// TwinCAT 3 PLC project Untitled1
// ProgramVersion: 3.1.4026.1+972e9c44872ad038b353624a861fd7e3244e9f75
// libraries:
//   Tc2_Standard, * (Beckhoff Automation GmbH)
//   Tc2_System, * (Beckhoff Automation GmbH)
//   Tc2_Utilities, * (Beckhoff Automation GmbH)
// project tree:
//   FolderControl/ E_FolderControlState.TcDUT, FB_FolderControl.TcPOU
//   FileWriter/ E_FileWriteState.TcDUT, FB_FileControl.TcPOU
//   / PlcTask.TcTTO
//   POUs/ MAIN.TcPOU
// real-time tasks:
//   TASK PlcTask: cycle T#10ms, priority 20, ADS port 350

CONFIGURATION Untitled1
    RESOURCE PLC ON TwinCAT3
        TASK PlcTask(INTERVAL := T#10ms, PRIORITY := 20);
        PROGRAM MAIN WITH PlcTask : MAIN;
    END_RESOURCE
END_CONFIGURATION

// ---- FolderControl/E_FolderControlState.TcDUT
{attribute 'qualified_only'}
{attribute 'strict'}
{attribute 'to_string'}
TYPE E_FolderControlState :
(
	init := 0,
	ReadyFindFolder := 10,
	FindFolder := 20,
	ReadyForCreateFolder := 100,
	CreateFolder := 110,
	Error := 999
);
END_TYPE

// ---- FileWriter/E_FileWriteState.TcDUT
{attribute 'qualified_only'}
{attribute 'strict'}
{attribute 'to_string'}
TYPE E_FileWriteState :
(
	init := 0,
	ReadyFileCreate := 5,
	FileOpen := 10, 
	FileWrite := 20, 
	FileClose := 30, 
	Error := 999
);
END_TYPE

// ---- POUs/MAIN.TcPOU
PROGRAM MAIN
VAR
	fbFolderControl : FB_FolderControl;
	sPath : T_MaxString := 'C:\Test\test2\test3';
	sFile : STRING;
	bStart: BOOL;
	bCheck: BOOL;
	
	step : INT;
	fbFileControl : FB_FileControl;
	sTest : T_MaxString;
END_VAR


IF bStart THEN
	bStart := FALSE;
	fbFolderControl.CreateFolder(sPath);
END_IF
IF bCheck THEN
	bCheck := FALSE;
	fbFolderControl.CheckFolder(sPath);
END_IF

fbFolderCOntrol.CyclicLogic();

CASE step OF
	0:
		;
	10:
		fbFileControl.OverwriteFile(sPath,ADR(sTest),LEN(sTest));
		step := 0;
	20:
		fbFileControl.AppendwriteFile(sPath,ADR(sTest),LEN(sTest));
		step := 0;
END_CASE
fbFileControl.CyclicLogit();

END_PROGRAM

// ---- FolderControl/FB_FolderControl.TcPOU
FUNCTION_BLOCK FB_FolderControl
VAR
	eState : E_FolderControlState;
	fbEnumFindFileEntry : FB_EnumFindFileEntry;
	fbCreateDir : FB_CreateDir;
	_CreateFolderPath : T_MAXSTRING;
	_CheckFolderPath : T_MAXSTRING;
	_FolderExist : BOOL;
	
	_Error : BOOL;
	_ErrorID : UDINT;
	_ErrorState : STRING(50);
	_AmsNetID : T_AmsNetID;
END_VAR

PROPERTY AmsNetId : T_AmsNetId
GET
AmsNetId := _AmsNetId;
END_GET
SET
_AmsNetId := AmsNetId;
END_SET
END_PROPERTY

{attribute 'monitoring':='call'}
PROPERTY Busy : BOOL
GET
Busy := NOT (eState = 0 OR eState = E_FolderControlState.Error);
END_GET
END_PROPERTY

METHOD CheckFolder : BOOL
VAR_INPUT
	sPath : T_MAXSTRING;
END_VAR
VAR
	i : INT;
END_VAR
IF Busy THEN
	RETURN;
END_IF
ResetStatus();

eState := E_FolderControlState.ReadyFindFolder;

MEMSET(ADR(_CheckFolderPath), 0, SIZEOF(_CheckFolderPath));

IF RIGHT(sPath,1) = '/' OR RIGHT(sPath,1) = '\' THEN
	sPath := Delete(sPath,1,LEN(sPath));
END_IF

FOR i:=0 TO LEN(sPath) BY 1 DO
	IF sPath[i] = 47 THEN 	// '/'
		_CheckFolderPath[i] := 92; 	// '\'
	ELSE
		_CheckFolderPath[i] := sPath[i];
	END_IF	
END_FOR

CheckFolder := TRUE;
END_METHOD

METHOD CreateFolder : BOOL
VAR_INPUT
	sPath : T_MAXSTRING;
END_VAR
VAR
	i : INT;
END_VAR
(*
	It only can create one more subfolder
	폴더 한번에 한개만 생성가능 즉, C:\Test\Test1\Test2 를 생성하고자 할때 Test1 폴더가 없으면 생성 불가
*)
IF Busy THEN
	RETURN;
END_IF
ResetStatus();

eState := E_FolderControlState.ReadyForCreateFolder;

MEMSET(ADR(_CreateFolderPath), 0, SIZEOF(_CreateFolderPath));

IF RIGHT(sPath,1) = '/' OR RIGHT(sPath,1) = '\' THEN
	sPath := Delete(sPath,1,LEN(sPath));
END_IF

FOR i:=0 TO LEN(sPath) BY 1 DO
	IF sPath[i] = 47 THEN 	// '/'
		_CreateFolderPath[i] := 92; 	// '\'
	ELSE
		_CreateFolderPath[i] := sPath[i];
	END_IF	
END_FOR

CreateFolder := TRUE;
END_METHOD

METHOD CyclicLogic
VAR_INPUT
END_VAR
CASE eState OF
	E_FolderControlState.init:
		;
		
	E_FolderControlState.ReadyFindFolder:
		fbEnumFindFileEntry(bExecute:= FALSE);
		fbEnumFindFileEntry.eCmd := E_EnumCmdType.eEnumCmd_First;
		_FolderExist := FALSE;
		eState := E_FolderControlState.FindFolder;
	
	E_FolderControlState.FindFolder:
		fbEnumFindFileEntry( 
			sPathName:= _CheckFolderPath, 
			bExecute:= TRUE);
		IF NOT fbEnumFindFileEntry.bBusy THEN
			IF fbEnumFindFileEntry.stFindFile.fileAttributes.bDirectory THEN
				_FolderExist := TRUE;
				eState := E_FolderControlState.init;
			END_IF
		END_IF
		
	E_FolderControlState.ReadyForCreateFolder:
		fbCreateDir(bExecute:= FALSE);
		eState := E_FolderControlState.CreateFolder;
		
	E_FolderControlState.CreateFolder:
		fbCreateDir(
			sNetId:= , 
			sPathName:= _CreateFolderPath,
			ePath:= E_OpenPath.PATH_GENERIC, 
			bExecute:= TRUE, 
			tTimeout:= , 
			bBusy=> , 
			bError=> , 
			nErrId=> );
		IF NOT fbCreateDir.bBusy THEN
			IF fbCreateDir.bError THEN
				_ErrorState := TO_STRING(E_FolderControlState.CreateFolder);
				eState := E_FolderControlState.Error;
				_ErrorID := fbCreateDir.nErrId;
			ELSE
				eState := E_FolderControlState.init;
			END_IF
		END_IF
	
	E_FolderControlState.Error:
		_Error := TRUE;
END_CASE
END_METHOD

{attribute 'monitoring':='variable'}
PROPERTY Error : BOOL
GET
Error := _Error;
END_GET
END_PROPERTY

{attribute 'monitoring':='variable'}
PROPERTY ErrorID : UDINT
GET
ErrorID := _ErrorID;
END_GET
END_PROPERTY

PROPERTY isFolderExist : BOOL
GET
isFolderExist := _FolderExist;
END_GET
END_PROPERTY

METHOD PRIVATE ResetStatus : BOOL
VAR_INPUT
END_VAR
_ErrorID := 0;
_Error := FALSE;
_ErrorState := '';
END_METHOD

END_FUNCTION_BLOCK

// ---- FileWriter/FB_FileControl.TcPOU
FUNCTION_BLOCK FB_FileControl
VAR
	fbFileWrite : FB_FileWrite;
	fbFileOpen : FB_FileOpen;
	fbFileClose : FB_FileClose;
	_Path : T_MAXSTRING;
	eState : E_FileWriteState;
	FileWriteMode : DWORD;
	
	_pSomethingToWrite : PVOID;
	_cbSomethingToWrite : UDINT;
	
	_Error : BOOL;
	_ErrorID : UDINT;
	_ErrorState : STRING(50);
	_AmsNetId : T_AmsNetId;
END_VAR

PROPERTY AmsNetId : T_AmsNetId
GET
AmsNetId := _AmsNetId;
END_GET
SET
_AmsNetId := AmsNetId;
END_SET
END_PROPERTY

METHOD AppendwriteFile : BOOL
VAR_INPUT
	sPathAndFileName : T_MAXSTRING; //Path and filename with file extension
	pSomethingtoWrite : PVOID;
	cbSomethingtoWrite : UDINT; 
END_VAR
IF Busy THEN
	RETURN;
END_IF
ResetStatus();
eState := E_FileWriteState.ReadyFileCreate;
_Path := sPathAndFileName;
FileWriteMode := FOPEN_MODEAPPEND OR FOPEN_MODETEXT;
_pSomethingtoWrite := pSomethingtoWrite;
_cbSomethingToWrite := cbSomethingtoWrite;
AppendwriteFile := TRUE;
END_METHOD

{attribute 'monitoring':='call'}
PROPERTY Busy : BOOL
GET
Busy := NOT(eState = 0 OR Error);
END_GET
END_PROPERTY

METHOD CyclicLogit
VAR_INST
	hFile : UINT;
END_VAR
CASE eState OF
	E_FileWriteState.Init:
		;
		
	E_FileWriteState.ReadyFileCreate:
		eState := E_FileWriteState.FileOpen;
		
	E_FileWriteState.FileOpen:
		fbFileOpen(sNetId:= _AmsNetID, 
					sPathName:= _Path, 
					nMode:= FileWriteMode, 
					bExecute:= TRUE,  
					hFile=> hFile);
		IF NOT fbFileOpen.bBusy THEN
			IF fbFileOpen.bError THEN
				eState := E_FileWriteState.Error;
				_ErrorID := fbFileOpen.nErrId;
				_ErrorState := TO_STRING(E_FileWriteState.FileOpen);
			ELSE
				eState := E_FileWriteState.FileWrite;
			END_IF
			fbFileOpen(bExecute := FALSE);	
		END_IF
		
	E_FileWriteState.FileWrite:
		fbFileWrite(sNetId:= _AmsNetID,
					hFile:= hFile, 
					pWriteBuff:= _pSomethingToWrite, 
					cbWriteLen:= _cbSomethingToWrite, 
					bExecute:= TRUE);
		IF NOT fbFileWrite.bBusy THEN
			IF fbFileWrite.bError THEN
				_ErrorID := fbFileWrite.nErrId;
				_ErrorState := TO_STRING(E_FileWriteState.FileWrite);
				eState := E_FileWriteState.Error;
			ELSE
				eState := E_FileWriteState.FileClose;	
			END_IF
			fbFileWrite(bExecute := FALSE);
		END_IF
		
	E_FileWriteState.FileClose:
		fbFileClose(sNetId:= _AmsNetID,
					hFile:= hFile, 
					bExecute:= TRUE);
		IF NOT fbFileClose.bBusy THEN
			IF fbFileClose.bError THEN
				eState := E_FileWriteState.Error;
				_ErrorID := fbFileClose.nErrId;
				_ErrorState := TO_STRING(E_FileWriteState.FileClose);
			ELSE
				eState := E_FileWriteState.Init;
			END_IF
			fbFileClose(bExecute := FALSE);
		END_IF
		
	E_FileWriteState.Error: 
		_Error := TRUE;
END_CASE
END_METHOD

{attribute 'monitoring':='variable'}
PROPERTY Error : BOOL
GET
Error := _Error;
END_GET
END_PROPERTY

{attribute 'monitoring':='variable'}
PROPERTY ErrorID : UDINT
GET
ErrorID := _ErrorID;
END_GET
END_PROPERTY

METHOD OverwriteFile : BOOL
VAR_INPUT
	sPathAndFileName : T_MAXSTRING; //Path and filename with file extension
	pSomethingtoWrite : PVOID;
	cbSomethingtoWrite : UDINT; //IF you put sizeof(string) they could be wrong data so, you should do LEN(string) 
END_VAR
IF Busy THEN
	RETURN;
END_IF
ResetStatus();
eState := E_FileWriteState.ReadyFileCreate;
_Path := sPathAndFileName;
FileWriteMode := FOPEN_MODEWRITE OR FOPEN_MODETEXT;
_pSomethingtoWrite := pSomethingtoWrite;
_cbSomethingToWrite := cbSomethingtoWrite;
OverWriteFile := TRUE;
END_METHOD

METHOD PRIVATE ResetStatus : BOOL
VAR_INPUT
END_VAR
_Error := FALSE;
_ErrorID := 0;
_ErrorState := '';
FileWriteMode := 0;

ResetStatus := TRUE;
END_METHOD

END_FUNCTION_BLOCK
